FUNCTION "Speed_SCL" : Void
{ S7_Optimized_Access := 'TRUE' }
VERSION : 0.1
   VAR_TEMP
      Speed : Real;
   END_VAR


BEGIN
	#Speed := 200;
END_FUNCTION

